{attribute 'qualified_only'}
{attribute 'strict'}
(*
TYPE Ds402_States :
(
	FSM_Ilegal := -2 ;
	FSM_NotReadyToSwitchOn := -1 ; 
	FSM_SwitchOnDisabled  := 0 ;
	FSM_ReadyToSwitchOn := 1;
	FSM_SwitchedOn := 2;
	FSM_OperationEnabled := 3 ;
	FSM_QuickStopActive := 4 ;
	FSM_FaultReactionActive := 5;
	FSM_Fault := 6 ; 
	FSM_Temporary_Fault := 7; 
);
END_TYPE
*)

(* stored: Version 1.1.0.1, ProductVersion 3.1.4024.6
   DUT Ds402_States: Id {e607a42e-9a9c-4743-ae85-756fb261249f} *)
